INTERFACE PUBLIC ActionStateCommands EXTENDS __System.IQueryInterface

METHOD PUBLIC StateComplete
END_METHOD

END_INTERFACE

(* stored: Version 1.1.0.1, ProductVersion 3.1.4026.18
   Itf ActionStateCommands: Id {a46ba3c8-bd22-0fe2-07b3-992c6e493e6e}
   Method StateComplete: Id {22da8347-601b-0ad6-2422-0601632470f0} *)
